TYPE ST_DcCurrent :
STRUCT
	
END_STRUCT
END_TYPE

(* stored: Version 1.1.0.1, ProductVersion 3.1.4022.3
   DUT ST_DcCurrent: Id {52d2de39-2b49-409e-bae8-96bd616c903f} *)
